TEXTLIST TextList_Dialogs
  0 = 'Control Gears - Commands'
  1 = 'Control Gears - Parameters'
  2 = 'Control Gears - Addressing'
  3 = 'Control Gears - Groups'
  4 = 'Control Gears - Scenes'
  5 = 'Control Gears - Memory Pages'
  6 = 'Control Gears - Set Fading'
  7 = 'Control Gears - Device Type 6 (LED)'
  8 = 'Control Devices - Parameters'
  9 = 'Control Devices - Addressing'
  10 = 'Control Devices - Device Type 1 (Push button)'
  11 = 'Control Devices - Device Type 2 (Absolute input)'
  12 = 'Control Devices - Device Type 3 (Occupancy sensor)'
  13 = 'Control Devices - Device Type 4 (Light sensor)'
  14 = 'Control Devices - Device Type 0 (Generic instance)'
  15 = 'Control Devices - Memory Pages'
  16 = 'Options KL6821'
   = ''
END_TEXTLIST

(* stored: Version 1.1.0.1, ProductVersion 3.1.4024.12
   TextList TextList_Dialogs: Id {549a1fb5-0049-4732-ae1c-91ef7c52241f} *)
